// TIA Portal V20 export
TYPE "type_emRelations_em5_cmStatus"
// stored: Access Published, Namespace Unit1
   STRUCT
      TransferPnPLeftSafetyPin : "LBC_typeDigitalSignalControlNode";
      TransferPnPLeftJRDetect : "LBC_typeDigitalSignalControlNode";
      TransferPnPRightSafetyPin : "LBC_typeDigitalSignalControlNode";
      TransferPnPRightJRDetect : "LBC_typeDigitalSignalControlNode";
      TransferPnPLeftAxisX : "LBC_typeAxis64PosControlNode";
      TransferPnPLeftAxisY : "LBC_typeAxis64PosControlNode";
      TransferPnPLeftAxisZ : "LBC_typeAxis64PosControlNode";
      TransferPnPRightAxisX : "LBC_typeAxis64PosControlNode";
      TransferPnPRightAxisY : "LBC_typeAxis64PosControlNode";
      TransferPnPRightAxisZ : "LBC_typeAxis64PosControlNode";
      TransferPnPLeftClampOpenClose : "LBC_typeTwoWayActuatorControlNode";
      TransferPnPRightClampOpenClose : "LBC_typeTwoWayActuatorControlNode";
   END_STRUCT;
END_TYPE
